FUNCTION_BLOCK WTAV_UINT (* Weighted Average *)
  (* Standard: 61499-1; Classification: Math; Function: Weighted average *)
  (* Version 0.2, 2004-09-25, JHC, Rockwell Automation, Deleted INIT, INITO; moved to fb.rt.math. *)
  (* Version 0.2, 2003-03-17, JHC, Rockwell Automation, Moved from fb.rt.omac to fb.rt.mach. *)
  (* Version 0.1, 2002-02-28, JHC, Rockwell Automation, Changed "=" to ":=", REAL_TO_INT to Java cast in ALGORITHM REQ. *)
  (* Version 0.0, 2001-04-14, JHC, Rockwell Automation, First XML version *)
  (* Compiler header: package fb.rt.math; *)
  (* Compiler Java Sun JDK 1.4.2 *)
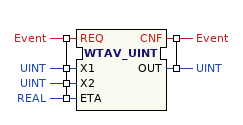
  EVENT_INPUT
    REQ WITH X1, X2, ETA; (* Normal Calculation *)
  END_EVENT
  EVENT_OUTPUT
    CNF WITH OUT; (* Execution Confirmation *)
  END_EVENT
  VAR_INPUT
    X1 : UINT; (* Value when ETA=0.0 *)
    X2 : UINT; (* Value when ETA=1.0 *)
    ETA : REAL;
  END_VAR
  VAR_OUTPUT
    OUT : UINT; (* ETA*X1+(1-ETA)*X2 *)
  END_VAR
  ALGORITHM REQ IN Java: (* Normally executed algorithm *)
OUT.value=(int)(X1.value+ETA.value*(X2.value-X1.value));
CNF.serviceEvent(this);
  END_ALGORITHM
END_FUNCTION_BLOCK
